(* IEC 61131-3 sources: AutomationLab/Support, 2 files *)

(* ---- G_Hardware.st ---- *)
// ============================================
// ФУНКЦИОНАЛЬНЫЙ БЛОК — обмен с аппаратурой
// Маппинг GVL physical I/O ↔ ConveyerData
// ============================================
FUNCTION_BLOCK G_Hardware
VAR_INPUT
END_VAR

VAR_OUTPUT
END_VAR

VAR_IN_OUT
    ConveyerData: ConveyerType; // данные конвейера
END_VAR

BEGIN
    // чтение физического сигнала датчика → данные конвейера
    ConveyerData.SensorA := GVL.DI_Sensor1;
    // команда вращения из данных конвейера → физический выход
    GVL.DO_ComMotor1 := ConveyerData.ComRotateLent;

END_FUNCTION_BLOCK

(* ---- G_Interface.st ---- *)
// ============================================
// ФУНКЦИОНАЛЬНЫЙ БЛОК — сопряжение с лампой оператора
// Маппинг ConveyerData ↔ GVL HMI
// ============================================
FUNCTION_BLOCK G_Interface
VAR_INPUT
END_VAR

VAR_OUTPUT
END_VAR

VAR_IN_OUT
    ConveyerData: ConveyerType; // данные конвейера
END_VAR

BEGIN
    // состояние конвейера → лампа на панели оператора
    GVL.DO_Lamp := ConveyerData.ComRotateLent;

END_FUNCTION_BLOCK
